RoboDK station: Example 1.2 - Linear rail & 2 fingers gripper Mouvements.rdk

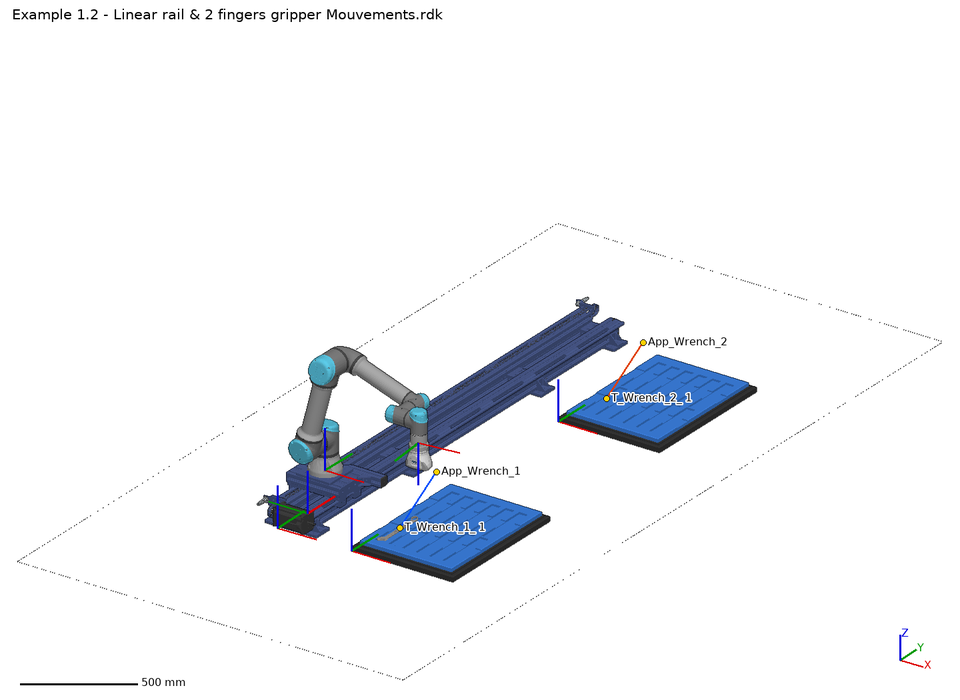
[picture v0: the station drawn from its stored meshes, robots at their saved joint values, targets as dots, program paths as lines]
Station Example 1.2 - 2 fingers gripper Station. Poses are relative to the parent item; angles as X-Y-Z fixed-axis rotations.
  - frame World at (0, 0, 0) mm
    - object Floor at (280, 1100, 0) mm, size 2000 x 4000 x 1 mm, geometry from plane_1m.sld
  - frame Linear Rail Base at (148.81, 12.71, 105) mm, rotated rx 0 ry 0 rz 90 deg
    - robot Linear Rail: 1 axes
        modified DH rows (alpha deg, a mm, theta deg, d mm): 0, 0, 0, 0 linear
        base shift (0, 0, 0) mm, rotated rx 0 ry 90 rz 0 deg
        joint limits [0] to [2100]; home [0]; saved at [150]
      - frame UR5e Base at (100, 85, 80) mm, rotated rx 0 ry 0 rz -90 deg
        - robot UR5e: 6 axes, payload 5 kg, reach 850 mm, repeatability 0.03 mm, weight 18.4 kg
            modified DH rows (alpha deg, a mm, theta deg, d mm): 0, 0, 0, 162.5; 90, 0, 180, 0; 0, 425, 0, 0; 0, 392.25, 0, 133.3; -90, 0, 0, 99.7; 90, 0, 180, 99.6
            joint limits [-360, -360, -360, -360, -360, -360] to [360, 360, 360, 360, 360, 360]; home [0, -90, -90, 0, 90, 0]; saved at [0, -104.57, -94.67, -70.76, 90, -95.16]
          - frame Schunk_Gripper Base at (0, 0, 0) mm
            - robot Schunk_Gripper: 1 axes
                joint limits [0] to [40]; home [40]; saved at [9]
          - tool Shunck_TCP, TCP at (0, 0, 190) mm
  - frame Frame Wrench 1 at (386.44, -2.63, 0) mm
    - target T_Wrench_1_ 1 (Cartesian target) at (100, 215, 50) mm, rotated rx 180 ry 0 rz 0 deg; joints [11.458, -119.591, -136.449, -13.961, 90, -78.542] of UR5e
    - target App_Wrench_1 (joint target) at (254.33, 266.39, 339.98) mm, rotated rx 180 ry 0 rz 5.16 deg; joints [0, -104.57, -94.67, -70.76, 90, -95.16] of UR5e
    - object Wrench Matrix at (25, 25, 10) mm, size 525 x 720 x 50 mm
    - object Wrench 1 at (100, 215, 65) mm, size 44.5 x 267.3 x 18.4 mm, geometry from Wrench.step
  - frame Frame Wrench 2 at (386.44, 1527.37, 0) mm
    - target T_Wrench_2_ 1 (Cartesian target) at (100, 215, 50) mm, rotated rx 180 ry 0 rz 0 deg; joints [11.458, -119.591, -136.449, -13.961, 90, -78.542] of UR5e
    - target App_Wrench_2 (joint target) at (254.33, 266.39, 339.98) mm, rotated rx 180 ry 0 rz 5.16 deg; joints [0, -104.57, -94.67, -70.76, 90, -95.16] of UR5e
    - object Wrench Matrix at (25, 25, 10) mm, size 525 x 720 x 50 mm
  - program ReplaceObjects (1 instructions, listed below)
  - folder RailPositions
  - folder GripperPositions
  - folder PickPrograms
    - program PickWrench (2 instructions, listed below)
    - program PickWrenchPos1 (6 instructions, listed below)
  - folder PlacePrograms
    - program PlaceWrench (2 instructions, listed below)
    - program PlaceWrenchPos1 (6 instructions, listed below)
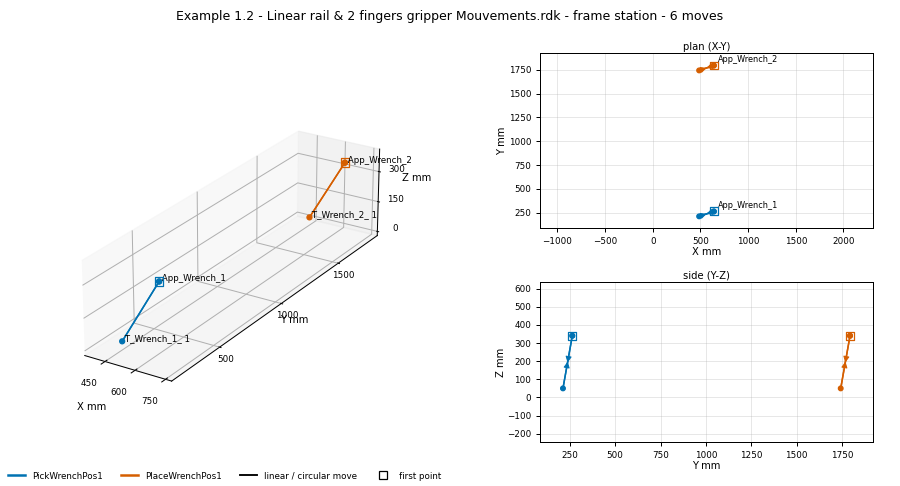
[picture p0: tool path of Example 1.2 - Linear rail & 2 fingers gripper Mouvements.rdk in frame station, 6 of 6 moves have a stored position in this frame; points joined in program order, loops and branches not executed]

--- program ReplaceObjects (robot UR5e) ---
  Replace objects

--- program PickWrench (robot UR5e) ---
  Call GripperPosPick
  Attach to Shunck_TCP

--- program PickWrenchPos1 (robot UR5e) ---
  Set Ref.: Frame Wrench 1
  Set Tool: Shunck_TCP
  MoveJ (App_Wrench_1)
  MoveL (T_Wrench_1_ 1)
  Call PickWrench
  MoveL (App_Wrench_1)

--- program PlaceWrench (robot UR5e) ---
  Call GripperPosOpen
  Detach from Shunck_TCP

--- program PlaceWrenchPos1 (robot UR5e) ---
  Set Ref.: Frame Wrench 2
  Set Tool: Shunck_TCP
  MoveJ (App_Wrench_2)
  MoveL (T_Wrench_2_ 1)
  Call PlaceWrench
  MoveL (App_Wrench_2)
